Fanuc KAREL source: w_d_uninit.kl

PROGRAM w_d_uninit
%NOLOCKGROUP
%UNINITVARS
VAR
  p : POSITION
  r : REAL
BEGIN
  WITH $SPEED = 500 MOVE TO p
  WITH $SPEED = r, $MOTYPE = LINEAR MOVE TO p
END w_d_uninit
